TYPE ExtendedAxisTyp  :
	STRUCT
		Basic_axis 	: Basic_axis_typ;
		MultiAxis 	: MultiAxis_typ;
		CyclicAxis	: CyclicAxis_typ;
		ParIDAccess	: ParIDAccess_Typ;
		VelocityCtrl: VelocityCtrl_typ;
	END_STRUCT
END_TYPE

(* stored: Version 1.1.0.1, ProductVersion 3.1.4024.3
   DUT ExtendedAxisTyp: Id {2a048db5-e06e-06b2-1721-2077e8d43366} *)
